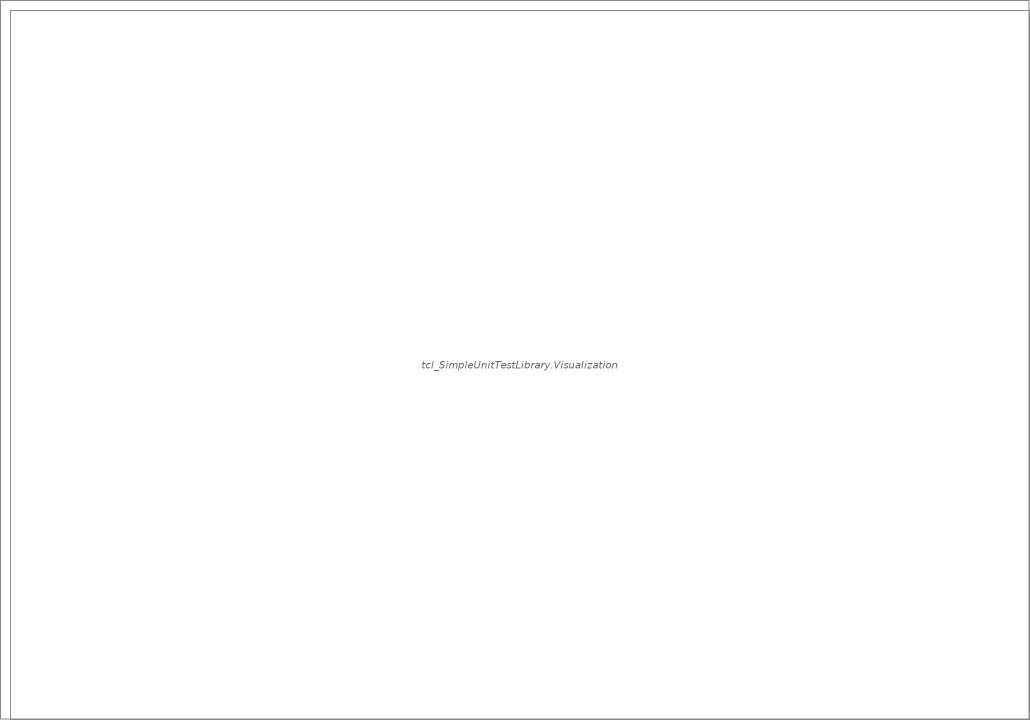
VISUALIZATION Visualization  // 1030x720
    Frame (10,10 1020x710)
        shows tcl_SimpleUnitTestLibrary.Visualization(TestRunner := PB_TestRunner.TestRunner, AssertionMessages := PB_TestRunner.TestRunner.AssertionMessages)
END_VISUALIZATION

(* stored: Version 1.1.0.1, ProductVersion 3.1.4024.6
   Visu Visualization: Id {0688adbe-6157-4178-b30c-453b69bd2559} *)
